// TIA Portal V20 export
// export: Created 2025-12-01T14:57:45.2358755Z, ExportSetting None, DisplayName Totally Integrated Automation Portal, DisplayVersion V20 Update 3, DisplayName TIA Portal Openness, DisplayVersion V20 Update 3, DisplayName TIA Portal Version Control Interface, DisplayVersion V20 Update 3, DisplayName STEP 7 Professional, DisplayVersion V20 Update 3, DisplayName STEP 7 Safety, DisplayVersion V20 Update 2, DisplayName WinCC Basic/Comfort/Advanced, DisplayVersion V20 Update 3, DisplayName WinCC Professional, DisplayVersion V20 Update 3, DisplayName WinCC Unified, DisplayVersion V20 Update 3
FUNCTION "FC784_Evento_INIR" : Void   // FC784, LAD
{ S7_Optimized_Access := 'FALSE' }
// stored: AutoNumber false, SetENOAutomatically false
   VAR_INPUT
      mensaje : Int;
   END_VAR
   VAR_TEMP
      numero : Int;
      numero_inicializacion : Int;
      pos_habi : Int;
      habi : String[2];
      ESTADO_HABI : Byte;
      ESTADO_HABI_BITS AT ESTADO_HABI : Array[1..8] of Bool;
      MENSAJE_EMI : String[50];
      Numero_string : String[1];
      atributo_habi : String[2];
      i : Int;
      longitud : Int;
   END_VAR
BEGIN

REGION Network 1 (SCL)
   // EXTRAEMOS EL VALOR DEL NUMERO DE LA INICIALIZACIÓN QUE TENEMOS QUE HABILITAR
   // 
   #numero := FIND(IN1 := "DB199_eventos_convertidos".evento[#mensaje], IN2 := '[NUME]');

   STRG_VAL(IN := "DB199_eventos_convertidos".evento[#mensaje],
            FORMAT := 0,
            P := (#numero + 6), // +6 por lo que ocupa el atributo ['SSCC]'
            OUT => #numero_inicializacion);

   // COMPROBAMOS LA VALIDED DEL NUMERO DE INICIALIZACIÓN. ACTUALMENTE EL MÁXIMO ES 8
   // 

   IF #numero_inicializacion > 8 THEN
       // formatear el mensaje de inicialización no posible
       // 

       #Numero_string := DELETE(IN := (INT_TO_STRING(IN := #numero_inicializacion)), L := 1, P := 1);
       // 
       #MENSAJE_EMI := CONCAT(IN1 := '{INI![NUME]', IN2 := #Numero_string, IN3 := '[HABI]NO[MOTI]NOOK', IN4 := "DB921_DATOS_FECHA_HORA".TIME_STAMP, IN5 := '}');

       REGION emision_mensaje
           // miramos donde tenemos que emitir el mensaje
           IF "ROUT_X_CONEX_JDT1" = FALSE THEN
               REGION buscar en JDT2                
                   FOR #i := 0 TO 100 BY 1 DO
                       #longitud := LEN("DB197_eventos_generados_routing_JDT2".evento[#i]);
                       IF #longitud = 0 THEN
                           "DB197_eventos_generados_routing_JDT2".evento[#i] := #MENSAJE_EMI;
                           RETURN;
                       END_IF;
                   END_FOR;
                   // si ha acabado el for sin encontrar sitio no puedo emititir y salgo de la funcion
                   RETURN;
               END_REGION
               ;
           ELSE
               REGION buscar en JDT1
                   FOR #i := 0 TO 100 BY 1 DO
                       #longitud := LEN("DB198_eventos_generados_routing_JDT1".evento[#i]);
                       IF #longitud = 0 THEN
                           "DB198_eventos_generados_routing_JDT1".evento[#i] := #MENSAJE_EMI;
                           RETURN;
                       END_IF;
                   END_FOR;
                   // si ha acabado el for sin encontrar sitio no puedo emititir y salgo de la funcion
                   RETURN;

               END_REGION
           END_IF;
       END_REGION
       ;
   END_IF;

   // EXTRAEMOS EL VALOR DEL ATRIBUTO HABI
   #pos_habi := FIND(IN1 := "DB199_eventos_convertidos".evento[#mensaje], IN2 := '[HABI]');

   #habi:=MID(IN:="DB199_eventos_convertidos".evento[#mensaje], L:=2, P:=#pos_habi+6);


   IF #habi = 'SI' THEN  //TENEMOS QUE HABILITAR LA INICIALIZACIÓN

       #ESTADO_HABI := "Estado_inicializacion";     // PRIMERO COGEMOS EL VALOR QUE TIENEN LAS MEMORIAS ACTUALENTE
       #ESTADO_HABI_BITS[#numero_inicializacion] := TRUE;
       "Estado_inicializacion" := #ESTADO_HABI;    //VOLVEMOS A VOLCAR EL ESTADO EN LA PALABRA GLOBAL

       // FORMATEAMOS EL MENSAJE



       #Numero_string := DELETE(IN := (INT_TO_STRING(IN := #numero_inicializacion)), L := 1, P := 1);

       #MENSAJE_EMI := CONCAT(IN1 := '{INI![NUME]', IN2 := #Numero_string, IN3 := '[HABI]SI', IN4 := "DB921_DATOS_FECHA_HORA".TIME_STAMP,IN5 := '}');

   ELSIF #habi = 'NO' THEN

       #ESTADO_HABI := "Estado_inicializacion"; // PRIMERO COGEMOS EL VALOR QUE TIENEN LAS MEMORIAS ACTUALENTE
       #ESTADO_HABI_BITS[#numero_inicializacion] := FALSE;
       "Estado_inicializacion" := #ESTADO_HABI;   //VOLVEMOS A VOLCAR EL ESTADO EN LA PALABRA GLOBAL

       // FORMATEAMOS EL MENSAJE



       #Numero_string := DELETE(IN := (INT_TO_STRING(IN := #numero_inicializacion)), L := 1, P := 1);

       #MENSAJE_EMI := CONCAT(IN1 := '{INI![NUME]', IN2 := #Numero_string, IN3 := '[HABI]NO', IN4 := "DB921_DATOS_FECHA_HORA".TIME_STAMP, IN5 := '}');

   ELSIF #habi = '??' THEN
       // MIRAMOS SI ESTÁ HABILITADO O NO PARA FORMATEAR EL MENSAJE
       #ESTADO_HABI := "Estado_inicializacion"; // PRIMERO COGEMOS EL VALOR QUE TIENEN LAS MEMORIAS ACTUALENTE

       IF #ESTADO_HABI_BITS[#numero_inicializacion] = TRUE THEN
           #atributo_habi := 'SI';
       ELSE
           #atributo_habi := 'NO';
       END_IF;


       // FORMATEAMOS EL MENSAJE


       #Numero_string := DELETE(IN := (INT_TO_STRING(IN := #numero_inicializacion)), L := 1, P := 1);

       #MENSAJE_EMI := CONCAT(IN1 := '{INI![NUME]', IN2 := #Numero_string, IN3 := '[HABI]',IN4:=#atributo_habi, IN5 := "DB921_DATOS_FECHA_HORA".TIME_STAMP, IN6 := '}');
       ;
   END_IF;


   REGION emision_mensaje
       // miramos donde tenemos que emitir el mensaje
       IF "ROUT_X_CONEX_JDT1" = FALSE THEN
           REGION buscar en JDT2                
               FOR #i := 0 TO 100 BY 1 DO
                       #longitud := LEN("DB197_eventos_generados_routing_JDT2".evento[#i]);
                       IF #longitud = 0 THEN
                           "DB197_eventos_generados_routing_JDT2".evento[#i]:=#MENSAJE_EMI;
                           RETURN;
                       END_IF;
                   END_FOR;
                   // si ha acabado el for sin encontrar sitio no puedo emititir y salgo de la funcion
                   RETURN;
               END_REGION
               ;
           ELSE
               REGION buscar en JDT1
                   FOR #i := 0 TO 100 BY 1 DO
                       #longitud := LEN("DB198_eventos_generados_routing_JDT1".evento[#i]);
                       IF #longitud = 0 THEN
                           "DB198_eventos_generados_routing_JDT1".evento[#i] := #MENSAJE_EMI;
                           RETURN;
                       END_IF;
                   END_FOR;
                   // si ha acabado el for sin encontrar sitio no puedo emititir y salgo de la funcion
                       RETURN;

               END_REGION
           END_IF;
   END_REGION
END_REGION
END_FUNCTION
